PROGRAM POU
VAR
	
	// Single line comment
	
	(* 
		Multiple line comment
	*)
		
	A AT %I* : BOOL := FALSE;
	B AT %I* : BOOL := FALSE;
	C AT %I* : BOOL := FALSE;
	D AT %Q* : BOOL := FALSE;
	
END_VAR

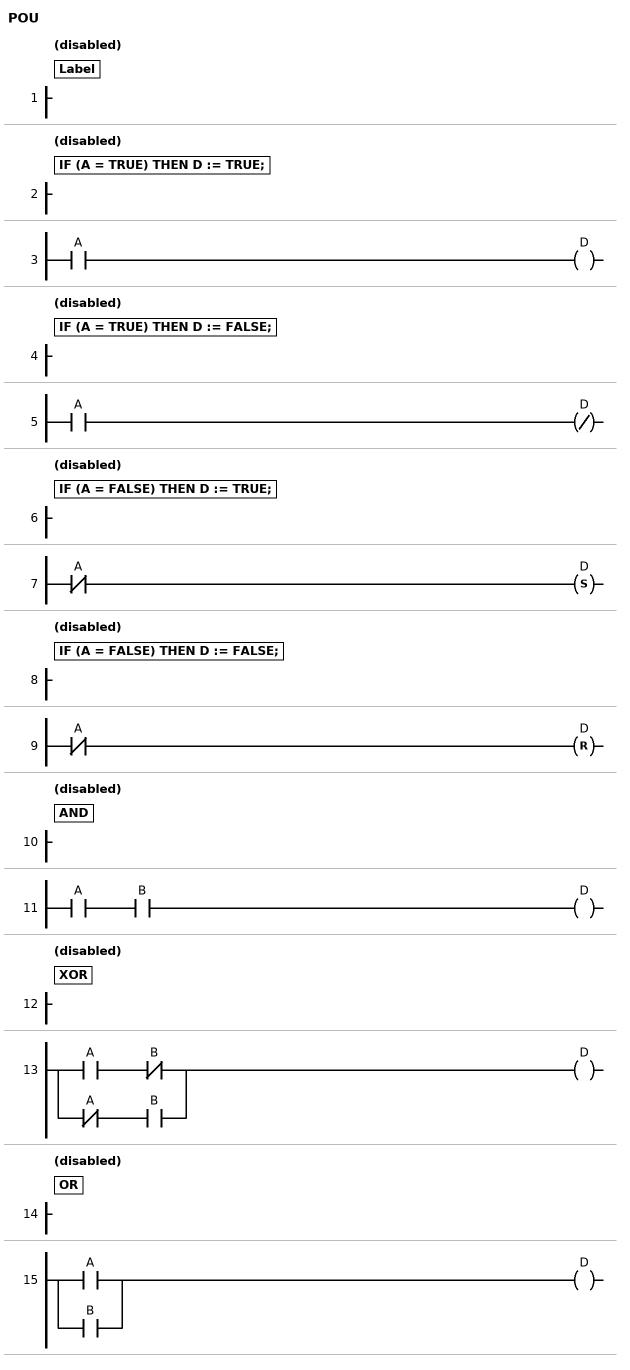
// NETWORK 1 (disabled)
// label: Label

// NETWORK 2 (disabled)
// label: IF (A = TRUE) THEN D := TRUE;

// NETWORK 3
D := A;

// NETWORK 4 (disabled)
// label: IF (A = TRUE) THEN D := FALSE;

// NETWORK 5
D := NOT A;

// NETWORK 6 (disabled)
// label: IF (A = FALSE) THEN D := TRUE;

// NETWORK 7
D S= NOT A;

// NETWORK 8 (disabled)
// label: IF (A = FALSE) THEN D := FALSE;

// NETWORK 9
D R= NOT A;

// NETWORK 10 (disabled)
// label: AND

// NETWORK 11
D := A AND B;

// NETWORK 12 (disabled)
// label: XOR

// NETWORK 13
D := A AND NOT B OR NOT A AND B;

// NETWORK 14 (disabled)
// label: OR

// NETWORK 15
D := A OR B;

END_PROGRAM

(* stored: Version 1.1.0.1, ProductVersion 3.1.4024.3
   POU POU: Id {bf5de3b6-88ba-4c75-ae2e-f538a68bd75e}, SpecialFunc None *)
